Universal Robots PolyScope program: rtde_control_loop_sigma_0920.urp

Program rtde_control_loop_sigma (installation=default directory=/home/ur/ursim-current/programs/programs createdIn=3.2.19275.0 lastSavedIn=5.6.0.90886 robotSerialNumber=20195399999)
Calibrated DH parameters: a=[0, -0.24355, -0.2132, 0, 0, 0]; d=[0.15185, 0, 0, 0.13105, 0.08535, 0.0921]; alpha=[1.570796, 0, 0, 1.570796, -1.570796, 0]; deltaTheta=[0, 0, 0, 0, 0, 0]
BeforeStart
  setp_p := p[0,0,0,0,0,0]
  setp_j := [0,0,0,0,0,0]
  inp_int_reg_0 := 0
  button_push_dis := 0.02
  Script: rtde_set_watchdog("input_int_register_0", 1, "PAUSE")
  Script: write_output_integer_register(0, 1)
Robot Program (runOnlyOnce=false)
  If inp_int_reg_0≟1
    'Valid pose received from client'
    inp_int_reg_0 := 0
    'Next time only with new position can be entered'
    If read_input_integer_register(1) ≟ 1
      MoveL speed 80 mm/s, acceleration 1200 mm/s^2 (useActiveTCP=true) feature=Base
        Waypoint Waypoint (Variable): variable=setp_p
    ElseIf read_input_integer_register(1)≟2
      'Pushing a button'
      current_pos := get_actual_tcp_pose()
      Script: current_pos[2] = current_pos[2] - button_push_dis
      MoveL speed 250 mm/s, acceleration 1200 mm/s^2 (useActiveTCP=true) feature=Base
        Waypoint Waypoint_1 (Variable): variable=current_pos
      Script: current_pos[2] = current_pos[2] + button_push_dis
      MoveL speed 250 mm/s, acceleration 1200 mm/s^2 (useActiveTCP=true) feature=Base
        Waypoint Waypoint_1 (Variable): variable=current_pos
    Else 
      MoveJ speed 60 deg/s, acceleration 80 deg/s^2 (useActiveTCP=true positionType=JointAngles) feature=Base
        Waypoint Waypoint (Variable): variable=setp_j
    'Confirm that move was executed'
    Script: write_output_integer_register(0, 0)
    'Wait until script acknowledges confirmation'
    Loop While (checkContinuously=false) expression=read_input_integer_register(0)≟1
      Script: sync()
    'Request next pose'
    Script: write_output_integer_register(0, 1)
  Script: sync()
Thread Thread_1 (runOnlyOnce=false)
  Loop Forever
    If read_input_integer_register(1) ≟ 1
      tmp_p := p[0,0,0,0,0,0]
      Script: tmp_p[0] = read_input_float_register(0)
      Script: tmp_p[1] = read_input_float_register(1)
      Script: tmp_p[2] = read_input_float_register(2)
      Script: tmp_p[3] = read_input_float_register(3)
      Script: tmp_p[4] = read_input_float_register(4)
      Script: tmp_p[5] = read_input_float_register(5)
      setp_p := tmp_p
    Else 
      tmp_j := [0,0,0,0,0,0]
      Script: tmp_j[0] = read_input_float_register(0)
      Script: tmp_j[1] = read_input_float_register(1)
      Script: tmp_j[2] = read_input_float_register(2)
      Script: tmp_j[3] = read_input_float_register(3)
      Script: tmp_j[4] = read_input_float_register(4)
      Script: tmp_j[5] = read_input_float_register(5)
      setp_j := tmp_j
    inp_int_reg_0 := read_input_integer_register(0)
    Script: sync()
